FUNCTION_BLOCK AX_BOOL_TO_X (* Composite FB for convert BOOL to AX *)
  (* Standard: 61499-2; Description: Copyright (c) 2024 HR Agrartechnik GmbH This program and the accompanying materials are made available under the terms of the Eclipse Public License 2.0 which is available at https://www.eclipse.org/legal/epl-2.0/ SPDX-License-Identifier: EPL-2.0 *)
  (* Version 1.0, 2024-04-24, Franz Höpfinger, HR Agrartechnik GmbH *)
  PACKAGE adapter::conversion::unidirectional;
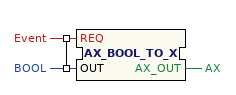
  EVENT_INPUT
    REQ WITH OUT; (* Request to Adapter *)
  END_EVENT
  VAR_INPUT
    OUT : BOOL;
  END_VAR
  PLUGS
    AX_OUT : adapter::types::unidirectional::AX; (* Adapter Output *)
  END_PLUGS
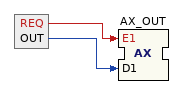
  EVENT_CONNECTIONS
    REQ TO AX_OUT.E1;
  END_CONNECTIONS
  DATA_CONNECTIONS
    OUT TO AX_OUT.D1;
  END_CONNECTIONS
END_FUNCTION_BLOCK
